// TwinCAT 3 PLC project XtesSxrPlc
// ProgramVersion: 3.1.4022.3
// libraries:
//   L2SI Vacuum Library, * (SLAC)
//   LCLS General, * (SLAC)
//   Tc2_Standard, * (Beckhoff Automation GmbH)
//   Tc2_System, * (Beckhoff Automation GmbH)
//   Tc2_Utilities, * (Beckhoff Automation GmbH)
//   Tc3_Module, * (Beckhoff Automation GmbH)
// project tree:
//   GVLs/ GVL_DEVICES.TcGVL (not stored), GVL_VARIABLES.TcGVL (not stored)
//   / PlcTask.TcTTO (not stored)
//   POUs/ MAIN.TcPOU, PRG_HEARTBEAT.TcPOU, PRG_PROTOTYPE.TcPOU (not stored)
// real-time tasks:
//   TASK PlcTask: cycle T#10ms, priority 20, ADS port 350
//   TASK SimTask: cycle T#5ms, priority 21, ADS port 351
// I/O:
//   DEVICE =+-AuxPS1-CPU/EtherCAT1, AmsNetId 5.45.6.154.2.1
//     =+-AuxPS1 [EK1100 EtherCAT Coupler (2A E-Bus)]
//       =+-DO1 [EL2794 4Ch. Dig. Output 24V AC/DC, 2A, short-circuit-proof]
//       =+-DI1 [EL1004 4Ch. Dig. Input 24V, 3ms]
//     =+-A1 [EP2338-0002 8 Ch. Dig. Input/Output 24V, 0,5A, M12]
//     =+-A2 [EP3174-0002 4Ch. Ana. Input +/-10V, 0-10V, 0/4-20mA configurable]
//     =+-A3 [EP2624-0002 4Ch. Relay Output, NO (125V AC / 30V DC)]
//   DEVICE Device 2 (EtherCAT Simulation), AmsNetId 5.45.6.154.3.1
//     =+-AuxPS1 // EK1100-0000-0018
//     =+-DO1 // EL2794-0000-0016
//     =+-DI1 // EL1004-0000-0019
//     =+-A1 // EP2338-0002-0023
//     =+-A2 // EP3174-0002-0023
//     =+-A3 // EP2624-0002-0019
// variable links:
//   ProtoSimPLC/ProtoSimPLC Instance <-> Device 2 (EtherCAT Simulation)/=+-A1
//     SimTask Inputs/GVL_DEVICES.stVgc_MR1K4_VGC_1.i_xSol <-> Channel 9/Output
//     SimTask Inputs/GVL_DEVICES.stVgc_TV2K4_VGC_1.i_xSol <-> Channel 13/Output
//     SimTask Outputs/GVL_DEVICES.stVgc_MR1K4_VGC_1.q_xClsLS <-> Channel 4/Input
//     SimTask Outputs/GVL_DEVICES.stVgc_MR1K4_VGC_1.q_xOpnLS <-> Channel 3/Input
//     SimTask Outputs/GVL_DEVICES.stVgc_TV2K4_VGC_1.q_xClsLS <-> Channel 8/Input
//     SimTask Outputs/GVL_DEVICES.stVgc_TV2K4_VGC_1.q_xOpnLS <-> Channel 7/Input
//   ProtoSimPLC/ProtoSimPLC Instance <-> Device 2 (EtherCAT Simulation)/=+-A2
//     SimTask Outputs/GVL_DEVICES.stMks275_TV2K4_GPI_1.q_iRawPress <-> AI Standard Channel 4/Value
//     SimTask Outputs/GVL_DEVICES.stMks500_TV2K4_GCC_1.q_iRawPress <-> AI Standard Channel 1/Value
//     SimTask Outputs/PRG_HEARTBEAT.heartbeat <-> AI Standard Channel 2/Value
//   ProtoSimPLC/ProtoSimPLC Instance <-> Device 2 (EtherCAT Simulation)/=+-A3
//     SimTask Inputs/GVL_DEVICES.stMks500_TV2K4_GCC_1.i_xHvOn <-> Channel 1/Output
//   ProtoSimPLC/ProtoSimPLC Instance <-> Device 2 (EtherCAT Simulation)/=+-DO1
//     SimTask Inputs/GVL_DEVICES.stGamPip_TV2KO_PIP_1.xOn <-> Channel 1/Output
//   XtesSxrPlc/XtesSxrPlc Instance <-> =+-AuxPS1-CPU/EtherCAT1/=+-A1
//     PlcTask Inputs/GVL_DEVICES.MR1K4_VGC_1.i_xClsLS <-> Channel 4/Input
//     PlcTask Inputs/GVL_DEVICES.MR1K4_VGC_1.i_xOpnLS <-> Channel 3/Input
//     PlcTask Inputs/GVL_DEVICES.TV2K4_VGC_1.i_xClsLS <-> Channel 8/Input
//     PlcTask Inputs/GVL_DEVICES.TV2K4_VGC_1.i_xOpnLS <-> Channel 7/Input
//     PlcTask Outputs/GVL_DEVICES.MR1K4_VGC_1.q_xOPN_DO <-> Channel 9/Output
//     PlcTask Outputs/GVL_DEVICES.TV2K4_VGC_1.q_xOPN_DO <-> Channel 13/Output
//   XtesSxrPlc/XtesSxrPlc Instance <-> =+-AuxPS1-CPU/EtherCAT1/=+-A2
//     PlcTask Inputs/GVL_DEVICES.TV2K4_GCC_1.i_iPRESS_R <-> AI Standard Channel 1/Value
//     PlcTask Inputs/GVL_DEVICES.TV2K4_GPI_1.i_iPRESS_R <-> AI Standard Channel 4/Value
//     PlcTask Inputs/PRG_HEARTBEAT.simHeartbeat <-> AI Standard Channel 2/Value
//   XtesSxrPlc/XtesSxrPlc Instance <-> =+-AuxPS1-CPU/EtherCAT1/=+-A3
//     PlcTask Outputs/GVL_DEVICES.TV2K4_GCC_1.q_xHV_DIS <-> Channel 1/Output
//   XtesSxrPlc/XtesSxrPlc Instance <-> =+-AuxPS1-CPU/EtherCAT1/=+-AuxPS1/=+-DI1
//     PlcTask Inputs/GVL_DEVICES.TV2KO_PIP_1.i_xSP_DI <-> Channel 4/Input
//   XtesSxrPlc/XtesSxrPlc Instance <-> =+-AuxPS1-CPU/EtherCAT1/=+-AuxPS1/=+-DO1
//     PlcTask Outputs/GVL_DEVICES.TV2KO_PIP_1.q_xHVEna_DO <-> Channel 1/Output

// ---- POUs/MAIN.TcPOU
PROGRAM MAIN
VAR
END_VAR

PRG_HEARTBEAT();
PRG_PROTOTYPE();

END_PROGRAM

// ---- POUs/PRG_HEARTBEAT.TcPOU
PROGRAM PRG_HEARTBEAT
VAR
	// for time logging
	fbTime : FB_LocalSystemTime := ( bEnable := TRUE, dwCycle := 1 );
	logTimer : TON := ( IN := TRUE, PT := T#1000ms );
	
	plcName : STRING[15];
	
	{attribute 'pytmc' := ' pv: simHeartbeat '}
	simHeartbeat AT %I* : UINT := 0;
	{attribute 'pytmc' := ' pv: plcHeartbeat '}
	plcHeartbeat : UDINT := 0;
	{attribute 'pytmc' := ' pv: plcInfo '}
	plcInfo : STRING[40];
	{attribute 'pytmc' := ' pv: plcLocalTime '}
	plcLocalTime : STRING[25];
END_VAR

plcHeartbeat := plcHeartbeat + 1;
IF plcHeartbeat > 4294967000
	THEN plcHeartbeat := 0;
END_IF

// get timestamp as string every second
fbTime();
logTimer( IN := fbTime.bValid );
IF logTimer.Q THEN
        logTimer( IN := FALSE ); logTimer( IN := fbTime.bValid );
        plcLocalTime := SYSTEMTIME_TO_STRING(fbTime.systemTime);
END_IF

// make an info string
plcName := 'Prototype PLC: ';
plcInfo := CONCAT(plcName, plcLocalTime);

END_PROGRAM
